(* IEC 61131-3 sources: Word/plc-course/14-analog-and-process-io/labs/starter, 3 files *)

(* ---- 14-1-analog-input.st ---- *)
(* Lab 14-1: FB_AnalogInput - raw counts to engineering units, with
   NAMUR NE43 fault detection, clamping, a first-order filter, a quality
   flag and substitute-value behaviour.
   Module 14 (Analog signals and process I/O). STARTER - the interface and the
   program that uses the block are done for you; write the body of
   FB_AnalogInput where it says TODO, then run:
     python3 tools/plctest.py 14-analog-and-process-io/labs/starter/14-1-analog-input.st

   Raw-count convention used by every lab in this module (Siemens style):
     Raw = 0     ->  4 mA   (bottom of the rated range)
     Raw = 27648 -> 20 mA   (top of the rated range)
     1 mA = 27648 / 16 = 1728 counts.
   Values outside 0..27648 are under- and over-range. The simulated card
   in this lab is linear over the whole INT range, so 0 mA reads -6912 and
   21 mA reads 29376. *)

FUNCTION_BLOCK FB_AnalogInput
  VAR_INPUT
    Raw        : INT;    (* raw count from the input card *)
    EuMin      : REAL;   (* engineering value at 4 mA (must be below EuMax) *)
    EuMax      : REAL;   (* engineering value at 20 mA *)
    FilterTime : TIME;   (* first-order filter time constant; T#0s = no filter *)
    FaultDelay : TIME;   (* signal must stay in a failure band this long before Fault *)
    UseSubst   : BOOL;   (* on Fault: TRUE = output SubstValue, FALSE = hold last good value *)
    SubstValue : REAL;   (* substitute value, engineering units *)
    CycleTime  : TIME;   (* interval of the task that calls this block *)
  END_VAR
  VAR_OUTPUT
    Current_mA : REAL;   (* loop current worked out from Raw: not filtered, not clamped *)
    Value      : REAL;   (* engineering value for the rest of the program *)
    Good       : BOOL;   (* TRUE while the loop current is inside the NE43 limits *)
    UnderRange : BOOL;   (* Fault, and the current is <= 3.6 mA: wire break, failure low *)
    OverRange  : BOOL;   (* Fault, and the current is >= 21.0 mA: short circuit, failure high *)
    Fault      : BOOL;   (* outside the NE43 limits for FaultDelay (= UnderRange OR OverRange) *)
  END_VAR
  VAR CONSTANT
    COUNTS_PER_MA : REAL := 1728.0;   (* 27648 counts / 16 mA *)
    FAIL_LOW_MA   : REAL := 3.6;      (* NE43: at or below = failure signal *)
    FAIL_HIGH_MA  : REAL := 21.0;     (* NE43: at or above = failure signal *)
  END_VAR
  VAR
    (* Suggested internal variables - add, rename or remove as you like. *)
    FaultTimer  : TON;    (* confirmation delay: signal outside the NE43 limits *)
    Filtered    : REAL;   (* filter state; also the last good value *)
    FilterReady : BOOL;   (* FALSE until the filter holds a real measurement *)
  END_VAR

  (* TODO: replace these placeholder lines with your logic (see the
     requirements in the Module 14 README, Lab 14-1). Suggested order:
       1. Raw -> Current_mA (convert to REAL first!)
       2. NE43 limits -> Good; then the FaultDelay -> Fault, UnderRange, OverRange
       3. Scale 4..20 mA to EuMin..EuMax and clamp
       4. First-order filter, fed only with good readings
       5. Value: substitute, hold or live *)
  Current_mA := 0.0;
  Value := 0.0;
  Good := FALSE;
  UnderRange := FALSE;
  OverRange := FALSE;
  Fault := FALSE;
END_FUNCTION_BLOCK

PROGRAM AnalogInputs
  VAR (* I/O - analog inputs, 0..27648 = 4..20 mA *)
    LT101_Raw AT %IW0 : INT;  (* LT-101 tank level transmitter: 0.0..4.0 m *)
    TT102_Raw AT %IW1 : INT;  (* TT-102 reactor temperature transmitter: -50..150 degC *)
  END_VAR
  VAR
    LT101 : FB_AnalogInput;   (* level: filtered, holds the last good value on a fault *)
    TT102 : FB_AnalogInput;   (* temperature: unfiltered, substitutes 150 degC on a fault *)
  END_VAR

  (* The program is complete: do not change these calls. *)
  LT101(Raw := LT101_Raw, EuMin := 0.0, EuMax := 4.0,
        FilterTime := T#2s, FaultDelay := T#1s,
        UseSubst := FALSE, SubstValue := 0.0, CycleTime := T#10ms);

  TT102(Raw := TT102_Raw, EuMin := -50.0, EuMax := 150.0,
        FilterTime := T#0s, FaultDelay := T#2s,
        UseSubst := TRUE, SubstValue := 150.0, CycleTime := T#10ms);
END_PROGRAM

CONFIGURATION Config0
  RESOURCE Res0 ON PLC
    TASK MainTask(INTERVAL := T#10ms, PRIORITY := 0);
    PROGRAM Inst0 WITH MainTask : AnalogInputs;
  END_RESOURCE
END_CONFIGURATION

(* ---- 14-2-analog-alarm.st ---- *)
(* Lab 14-2: FB_AnalogAlarm - HH/H/L/LL process alarms with a deadband
   (hysteresis) and an on-delay, so a noisy signal cannot make them chatter.
   Module 14 (Analog signals and process I/O). STARTER - the interface and the
   program that uses the block are done for you; write the body of
   FB_AnalogAlarm where it says TODO, then run:
     python3 tools/plctest.py 14-analog-and-process-io/labs/starter/14-2-analog-alarm.st

   Tip: four limits behave the same way (two mirrored). You may write a
   small helper FUNCTION_BLOCK for ONE limit and use four instances of it.
   MATIEC cannot make an array of FB instances, so declare four variables.
   Don't call an input "Limit": LIMIT is a standard function name. *)

FUNCTION_BLOCK FB_AnalogAlarm
  VAR_INPUT
    PV       : REAL;   (* process value, engineering units *)
    HH_Limit : REAL;   (* high-high limit *)
    H_Limit  : REAL;   (* high limit *)
    L_Limit  : REAL;   (* low limit *)
    LL_Limit : REAL;   (* low-low limit *)
    Deadband : REAL;   (* engineering units, the same for all four limits *)
    OnDelay  : TIME;   (* the same for all four limits; each needs its own timer *)
  END_VAR
  VAR_OUTPUT
    HH : BOOL;         (* PV >= HH_Limit for OnDelay; clears below HH_Limit - Deadband *)
    H  : BOOL;         (* PV >= H_Limit  for OnDelay; clears below H_Limit  - Deadband *)
    L  : BOOL;         (* PV <= L_Limit  for OnDelay; clears above L_Limit  + Deadband *)
    LL : BOOL;         (* PV <= LL_Limit for OnDelay; clears above LL_Limit + Deadband *)
  END_VAR
  VAR
    (* Add your internal variables here (timers, helper FB instances ...). *)
    HH_Timer : TON;
  END_VAR

  (* TODO: replace these placeholder lines with your logic (see the
     requirements in the Module 14 README, Lab 14-2). *)
  HH := FALSE;
  H := FALSE;
  L := FALSE;
  LL := FALSE;
END_FUNCTION_BLOCK

PROGRAM AlarmDemo
  VAR (* process values: in a real program these come from FB_AnalogInput
         (Lab 14-1). Here the test writes them directly. *)
    Level    : REAL;   (* LT-201 tank level, % *)
    Pressure : REAL;   (* PT-202 header pressure, bar *)
  END_VAR
  VAR
    LevelAlm : FB_AnalogAlarm;
    PressAlm : FB_AnalogAlarm;
  END_VAR

  (* The program is complete: do not change these calls. *)
  LevelAlm(PV := Level, HH_Limit := 90.0, H_Limit := 80.0, L_Limit := 20.0, LL_Limit := 10.0,
           Deadband := 2.0, OnDelay := T#3s);

  PressAlm(PV := Pressure, HH_Limit := 8.0, H_Limit := 7.0, L_Limit := 2.0, LL_Limit := 1.0,
           Deadband := 0.2, OnDelay := T#0s);
END_PROGRAM

CONFIGURATION Config0
  RESOURCE Res0 ON PLC
    TASK MainTask(INTERVAL := T#10ms, PRIORITY := 0);
    PROGRAM Inst0 WITH MainTask : AlarmDemo;
  END_RESOURCE
END_CONFIGURATION

(* ---- 14-3-sump-pump.st ---- *)
(* Lab 14-3: Sump pump level control - a pump-down on/off controller with
   hysteresis, a high-level alarm, an independent low-low float for dry-run
   protection, pump fault handling, and a level-transmitter fault.
   Module 14 (Analog signals and process I/O). STARTER - the declarations are
   done for you; write the logic where it says TODO, then run:
     python3 tools/plctest.py 14-analog-and-process-io/labs/starter/14-3-sump-pump.st

   TRAINING EXERCISE ONLY. The low-low float trip here is ordinary control
   logic in a standard PLC, not a designed safety function (Module 20).

   Raw-count convention: 0..27648 = 4..20 mA, 1728 counts per mA.
   LT-301 range 0.0..4.0 m, so 1 m = 6912 counts.

   Reuse your work: paste your FB_AnalogInput from Lab 14-1 (and, if you
   like, FB_AnalogAlarm from Lab 14-2) ABOVE the PROGRAM, then declare an
   instance of it below. MATIEC compiles one file, so the blocks must be
   in this file. *)

PROGRAM SumpPump
  VAR (* I/O *)
    LT301_Raw     AT %IW0   : INT;   (* LT-301 sump level: 0..27648 = 4..20 mA = 0.0..4.0 m *)
    LSLL302_NC    AT %IX0.0 : BOOL;  (* low-low float, NC: TRUE while water is above it *)
    PumpRunFb     AT %IX0.1 : BOOL;  (* pump contactor auxiliary contact: TRUE = pulled in *)
    PumpOL_NC     AT %IX0.2 : BOOL;  (* motor overload relay, NC: TRUE = healthy *)
    ResetPB       AT %IX0.3 : BOOL;  (* fault reset push-button, NO *)
    PumpRun       AT %QX0.0 : BOOL;  (* pump contactor coil *)
    HighLevelAlm  AT %QX0.1 : BOOL;  (* high sump level alarm *)
    LowLowAlm     AT %QX0.2 : BOOL;  (* low-low float operated (latched) *)
    PumpFaultAlm  AT %QX0.3 : BOOL;  (* pump fault: overload or no run feedback (latched) *)
    LevelFaultAlm AT %QX0.4 : BOOL;  (* LT-301 signal outside the NE43 limits *)
  END_VAR
  VAR
    Level : REAL;                    (* sump level in m, for the HMI *)
  END_VAR
  VAR CONSTANT
    START_LEVEL    : REAL := 2.0;    (* pump starts at or above this level, m *)
    STOP_LEVEL     : REAL := 1.0;    (* pump stops at or below this level, m *)
    HIGH_ALM_LEVEL : REAL := 3.0;    (* high level alarm limit, m *)
    HIGH_ALM_DB    : REAL := 0.1;    (* high level alarm deadband, m *)
  END_VAR
  VAR
    (* Suggested internal variables - add, rename or remove as you like.
       For example: LT301 : FB_AnalogInput; (after pasting the block) *)
    HighAlmTimer : TON;              (* 5 s on-delay for the high level alarm *)
    FbTimer      : TON;              (* 2 s run-feedback supervision *)
    ResetEdge    : R_TRIG;           (* reset acts on the press *)
    Demand       : BOOL;             (* the level controller wants the pump on *)
  END_VAR

  (* TODO: replace these placeholder lines with your logic (see the
     requirements in the Module 14 README, Lab 14-3). *)
  Level := 0.0;
  PumpRun := FALSE;
  HighLevelAlm := FALSE;
  LowLowAlm := FALSE;
  PumpFaultAlm := FALSE;
  LevelFaultAlm := FALSE;
END_PROGRAM

CONFIGURATION Config0
  RESOURCE Res0 ON PLC
    TASK MainTask(INTERVAL := T#10ms, PRIORITY := 0);
    PROGRAM Inst0 WITH MainTask : SumpPump;
  END_RESOURCE
END_CONFIGURATION
